(* IEC 61131-3 sources: repolevel_ST_code_completion/extract_code/重型运输系统/modbus/FUN, 16 files *)

(* ---- DataReverse_cmdReverse.st ---- *)
FUNCTION cmdReverse : TargetDirect
VAR_INPUT
	input		:TargetDirect;
END_VAR

IF input = TargetDirect.extend THEN
	cmdReverse := TargetDirect.retract;
END_IF
IF input = TargetDirect.retract THEN
	cmdReverse := TargetDirect.extend;
END_IF

(* ---- percentCalc.st ---- *)
FUNCTION percentCalc : REAL
VAR_INPUT
	level		:INT;	//1->地轨	2->天轨
	idx			:INT;	//挡板索引编号
END_VAR
VAR
	c			:REAL;
	p			:REAL;
END_VAR

//伸出百分比计算
CASE level OF
	1:
		IF gDev.grd[idx].sensor.position < 3 THEN
			RETURN;
		END_IF
		c := gDev.grd[idx].sensor.position - gDev.grd[idx].sensor.retractVal;
		p := gDev.grd[idx].sensor.extendVal - gDev.grd[idx].sensor.retractVal;
		percentCalc := c * 100 / p;
	2:
		IF gDev.sky[idx].sensor.position < 3 THEN
			RETURN;
		END_IF
		c := gDev.sky[idx].sensor.position - gDev.sky[idx].sensor.retractVal;
		p := gDev.sky[idx].sensor.extendVal - gDev.sky[idx].sensor.retractVal;
		percentCalc := c * 100 / p;
END_CASE

(* ---- setButtonByDirect.st ---- *)
FUNCTION setButtonByDirect : BOOL
VAR_INPUT
	level		:INT;	//1->地轨	2->天轨
	idx			:INT;	//挡板索引编号
	direct		:TargetDirect;
END_VAR
VAR
END_VAR
//	本函数用于根据输入参数 操作UI界面的按钮变量
CASE level OF
	1:
		IF idx = 0 OR idx > 10 THEN		//参数校验
			RETURN;
		END_IF
		CASE direct OF
			TargetDirect.extend:
				gUI.grd[idx].btnStop := FALSE;
				gUI.grd[idx].btnExtend := TRUE;
				gUI.grd[idx].btnRetract := FALSE;
			TargetDirect.retract:
				gUI.grd[idx].btnStop := FALSE;
				gUI.grd[idx].btnExtend := FALSE;
				gUI.grd[idx].btnRetract := TRUE;
			TargetDirect.stop:
				gUI.grd[idx].btnStop := FALSE;
				gUI.grd[idx].btnExtend := FALSE;
				gUI.grd[idx].btnRetract := FALSE;
		END_CASE
	2:
		IF idx > 10 THEN		//参数校验
			RETURN;
		END_IF
		CASE direct OF
			TargetDirect.extend:
				gUI.sky[idx].btnStop := FALSE;
				gUI.sky[idx].btnExtend := TRUE;
				gUI.sky[idx].btnRetract := FALSE;
			TargetDirect.retract:
				gUI.sky[idx].btnStop := FALSE;
				gUI.sky[idx].btnExtend := FALSE;
				gUI.sky[idx].btnRetract := TRUE;
			TargetDirect.stop:
				gUI.sky[idx].btnStop := FALSE;
				gUI.sky[idx].btnExtend := FALSE;
				gUI.sky[idx].btnRetract := FALSE;
		END_CASE

END_CASE;

(* ---- updateDevStatus.st ---- *)
FUNCTION updateDevStatus : DevStatus
VAR_INPUT
	level		:INT;		//1->地轨	2->天轨
	idx			:INT;		//挡板索引编号
	errorVal	:REAL;		//误差范围
END_VAR
VAR
	extendVal	:REAL;		//伸出值
	retractVal	:REAL;		//缩回到位值
	nowVal		:REAL;		//当前值
	stat		:DevStatus;	//设备状态
END_VAR

(* 本函数用于根据设备的标定伸出/缩回值以及当前位置
** 判断该缸体是否处于伸出/缩回到位状态，如果到位更新参数
*)

stat := DevStatus.unknown;	//初始化状态量
CASE level OF
	1:
		extendVal := gDev.grd[idx].sensor.extendVal;
		retractVal := gDev.grd[idx].sensor.retractVal;
		nowVal := gDev.grd[idx].sensor.position;
		stat := gDev.grd[idx].state;
	2:
		extendVal := gDev.sky[idx].sensor.extendVal;
		retractVal := gDev.sky[idx].sensor.retractVal;
		nowVal := gDev.sky[idx].sensor.position;
		stat := gDev.sky[idx].state;
END_CASE

IF nowVal > 1 THEN
	IF nowVal < retractVal + errorVal THEN
		stat := DevStatus.retracted;
	ELSIF nowVal > extendVal - errorVal THEN
		stat := DevStatus.extended;
	ELSE
		IF stat <> DevStatus.runing THEN
			stat := DevStatus.error;
		END_IF
	END_IF
ELSE
	stat := DevStatus.unknown;
END_IF

CASE level OF
	1:
		gDev.grd[idx].state := stat;
	2:
		gDev.sky[idx].state := stat;
END_CASE

updateDevStatus := stat;

(* ---- CommandExecutor.st ---- *)
FUNCTION_BLOCK CommandExecutor
VAR_INPUT
	level		:INT;			//1->地轨	2->天轨
	idx			:INT;			//挡板索引编号
	percent		:REAL;			//比例阀百分比 传入-100~+100
END_VAR
VAR_OUTPUT
END_VAR
VAR
END_VAR

IF percent > 0 THEN
	CASE level OF
		1:
			gController.grd[idx].extendPercent := REAL_TO_WORD(percent * 65535 / 100);
			gController.grd[idx].retractPercent := 0;
		2:
			gController.sky[idx].extendPercent := REAL_TO_WORD(percent * 65535 / 100);
			gController.sky[idx].retractPercent := 0;
	END_CASE
ELSE
	CASE level OF
		1:
			gController.grd[idx].extendPercent := 0;
			gController.grd[idx].retractPercent := REAL_TO_WORD(ABS(percent) * 65535 / 100);
		2:
			gController.sky[idx].extendPercent := 0;
			gController.sky[idx].retractPercent := REAL_TO_WORD(ABS(percent) * 65535 / 100);
	END_CASE
END_IF

(* ---- CommandExecutor0.st ---- *)
FUNCTION_BLOCK CommandExecutor0
VAR_INPUT
	level		:INT;			//1->地轨	2->天轨
	idx			:INT;			//挡板索引编号
	direct		:TargetDirect;	//方向
	percent		:REAL;			//比例阀百分比 传入0-100
END_VAR
VAR_OUTPUT
END_VAR
VAR
END_VAR

CASE direct OF
	TargetDirect.extend:
		CASE level OF
			1:
				gController.grd[idx].extendPercent := REAL_TO_WORD(percent * 65535 / 100);
				gController.grd[idx].retractPercent := 0;
			2:
				gController.sky[idx].extendPercent := REAL_TO_WORD(percent * 65535 / 100);
				gController.sky[idx].retractPercent := 0;
		END_CASE
	TargetDirect.retract:
		CASE level OF
			1:
				gController.grd[idx].extendPercent := 0;
				gController.grd[idx].retractPercent := REAL_TO_WORD(percent * 65535 / 100);
			2:
				gController.sky[idx].extendPercent := 0;
				gController.sky[idx].retractPercent := REAL_TO_WORD(percent * 65535 / 100);
		END_CASE
	TargetDirect.stop:
		CASE level OF
			1:
				gController.grd[idx].extendPercent := 0;
				gController.grd[idx].retractPercent := 0;
			2:
				gController.sky[idx].extendPercent := 0;
				gController.sky[idx].retractPercent := 0;
		END_CASE

	ELSE
		CASE level OF
			1:
				gController.grd[idx].extendPercent := 0;
				gController.grd[idx].retractPercent := 0;
			2:
				gController.sky[idx].extendPercent := 0;
				gController.sky[idx].retractPercent := 0;
		END_CASE

END_CASE

(* ---- DataReverse.st ---- *)
FUNCTION_BLOCK DataReverse
VAR_INPUT
END_VAR
VAR_OUTPUT
END_VAR
VAR
END_VAR

(* ---- fileSave.st ---- *)
FUNCTION_BLOCK fileSave
VAR_INPUT
	filePath 	:STRING;
	intervalt	:INT;
END_VAR
VAR
	lineCount	: INT;
	fileHandle  : DWORD;
	fileName	: STRING;
END_VAR
VAR_OUTPUT
END_VAR

(* ---- fileSave_close.st ---- *)
FUNCTION_BLOCK fileSave
VAR_INPUT
	filePath 	:STRING;
	intervalt	:INT;
END_VAR
VAR
	lineCount	: INT;
	fileHandle  : DWORD;
	fileName	: STRING;
END_VAR
VAR_OUTPUT
END_VAR

IF fileHandle <> 0 THEN
	SysFileClose(hFile := fileHandle);
	fileHandle := 0;
END_IF

(* ---- fileSave_createDir.st ---- *)
FUNCTION_BLOCK fileSave
VAR_INPUT
	filePath 	:STRING;
	devName		: STRING ;
	intervalt	:INT;
END_VAR
VAR
	lineCount	: INT;
	fileHandle  : DWORD;
	fileName	: STRING;
	filePath1	:STRING;
END_VAR
VAR_OUTPUT
END_VAR

filePath1 := FilePath;
filePath1 := concat(filePath1,'/');
filePath1 := concat(filePath1,devName);
SysDirCreate2(filePath1, TRUE);

(* ---- fileSave_new.st ---- *)
FUNCTION_BLOCK fileSave
VAR_INPUT
	filePath 	:STRING;
	intervalt	:INT;
	devName		: STRING ;
END_VAR
VAR
	lineCount	: INT;
	fileHandle  : DWORD;
	fileName	: STRING;
	fileHandle0 : DWORD;
	datetime	: DATE_AND_TIME;
	UdIntms 	: UDINT;
	UdMsOffset  : UDINT;
	DTimer_Str  : STRING;
	uiYear 		: UINT;
    uiMonth 	: UINT;
    uiDay 		: UINT;
    uiHour 		: UINT;
    uiMinute 	: UINT;
    uiSecond 	: UINT;
	uiMsSecond	: UINT;

	S_Time64		:  SysTime64;
	STT			:  CurTimeEx;
	S_Time			:  SystemTimeDate;
	Time_Str		:  STRING;
	F_err		: DWORD;
	F_HANDL		: DWORD;
END_VAR
VAR_OUTPUT
END_VAR

	STT(SystemTime:= S_Time64, TimeDate:= S_Time);
	Time_Str :='';
	Time_Str := concat(Time_Str,UINT_TO_STRING(S_Time.Year));
	Time_Str := concat(Time_Str,'-');
	Time_Str := concat(Time_Str,UINT_TO_STRING(S_Time.Month));
	Time_Str := concat(Time_Str,'-');
	Time_Str := concat(Time_Str,UINT_TO_STRING(S_Time.Day));
	Time_Str := concat(Time_Str,'_');
	Time_Str := concat(Time_Str,UINT_TO_STRING(S_Time.Hour));
	Time_Str := concat(Time_Str,'-');
	Time_Str := concat(Time_Str,UINT_TO_STRING(S_Time.Minute));
	Time_Str := concat(Time_Str,'-');
	Time_Str := concat(Time_Str,UINT_TO_STRING(S_Time.Second));
	Time_Str := concat(Time_Str,'_');
	Time_Str := concat(Time_Str,UINT_TO_STRING(S_Time.Milliseconds));

	fileName := FilePath;
	fileName := concat(fileName,'/');
	fileName := concat(fileName,devName);

	fileName := concat(fileName,'/');
	fileName := concat(fileName,devName);
	fileName := concat(fileName,'-');
	fileName := concat(fileName,Time_Str);
    fileName := concat(fileName,'.txt');

	fileHandle := SysFileOpen(szFile:= fileName, am:=ACCESS_MODE.AM_WRITE, pResult:= ADR(F_err));
	lineCount := -1;
	//fileHandle := SysFileOpen(szFile:= fileName, am:=ACCESS_MODE.AM_APPEND, pResult:= ADR(F_err));

(* ---- fileSave_write.st ---- *)
FUNCTION_BLOCK fileSave
VAR_INPUT
	filePath 	:STRING;
	intervalt	:INT;
	positionInt 	:INT;
	speedInt 		:INT;
	stateInt		:INT;
END_VAR
VAR
	lineCount	: INT;
	fileHandle  : DWORD;
	fileName	: STRING;
	data		: STRING;
	F_err		: DWORD;
	tempInt		: INT;
END_VAR
VAR_OUTPUT
END_VAR

IF fileHandle <> 0 THEN
	lineCount := lineCount + 1;
	tempInt	:= lineCount * intervalt;
	data := INT_TO_STRING(lineCount);
	data := concat(data,'$T$T');
	data := concat(data, INT_TO_STRING(tempInt));
	IF tempInt < 1000 THEN
		data := concat(data,'$T');
	END_IF
	data := concat(data,'$T$T');
	data := concat(data,INT_TO_STRING(positionInt));
	data := concat(data,'$T');
	data := concat(data,INT_TO_STRING(speedInt));
	data := concat(data,'$T');
	data := concat(data,INT_TO_STRING(stateInt));
	data := concat(data,'$R');

	SysFileWrite(hFile:=fileHandle , pbyBuffer:= ADR(data) , ulSize:= DINT_TO_DWORD(SysStrLen(data)) , pResult:= ADR(F_err));		// 写入数据

END_IF

(* ---- mdbsLogicToPhy.st ---- *)
FUNCTION_BLOCK mdbsLogicToPhy	//modbus华中挡板地址编号对应本地索引编号
VAR_INPUT
	section		:INT;	//区域限定 1:skyExt, 2:skyRet, 3:grdExt, 4:grdRet)
	lgcIdx		:INT;	//华中对应的地址	10,14{1..10}  17,20{1..11}
END_VAR
VAR_OUTPUT
	level		:INT;	//1->地轨	2->天轨
	phyIdx		:INT;	//内存物理地址对应数组索引
	direct		:TargetDirect;
END_VAR
VAR
END_VAR

(**
 * 将华中指令解析为要动作挡板的标号
 * (level:1->地轨	2->天轨)(phyIdx:内存物理地址对应数组索引)
 *)
CASE section OF
	1://区域限定1:skyExtend)
		level := 2;
		direct := TargetDirect.extend;
		CASE lgcIdx OF
			1:	phyIdx := 1;		//横1	->	sky1
			2:	phyIdx := 3;		//横2	->	sky3
			3:	phyIdx := 4;		//横3	->	sky4
			4:	phyIdx := 5;		//横4	->	sky5
			5:	phyIdx := 6;		//横5	->	sky6
			6:	phyIdx := 8;		//横6	->	sky8
			7:	phyIdx := 9;		//横7	->	sky9
			8:	phyIdx := 10;		//横8	->	sky10
			9:	phyIdx := 2;		//纵1	->	sky2
			10:	phyIdx := 7;		//纵2	->	sky7
			11:	phyIdx := 0;		//起竖	->	sky0
		END_CASE

	2://区域限定2:skyRetract)
		level := 2;
		direct := TargetDirect.retract;
		CASE lgcIdx OF
			1:	phyIdx := 1;		//横1	->	sky1
			2:	phyIdx := 3;		//横2	->	sky3
			3:	phyIdx := 4;		//横3	->	sky4
			4:	phyIdx := 5;		//横4	->	sky5
			5:	phyIdx := 6;		//横5	->	sky6
			6:	phyIdx := 8;		//横6	->	sky8
			7:	phyIdx := 9;		//横7	->	sky9
			8:	phyIdx := 10;		//横8	->	sky10
			9:	phyIdx := 2;		//纵1	->	sky2
			10:	phyIdx := 7;		//纵2	->	sky7
			11:	phyIdx := 0;		//起竖	->	sky0
		END_CASE

	3://区域限定3:grdExtend)
		level := 1;
		direct := TargetDirect.extend;
		CASE lgcIdx OF
			1:	phyIdx := 1;		//横1	->	grd1
			2:	phyIdx := 3;		//横2	->	grd3
			3:	phyIdx := 4;		//横3	->	grd4
			4:	phyIdx := 5;		//横4	->	grd5
			5:	phyIdx := 6;		//横5	->	grd6
			6:	phyIdx := 8;		//横6	->	grd8
			7:	phyIdx := 9;		//横7	->	grd9
			8:	phyIdx := 10;		//横8	->	grd10
			9:	phyIdx := 2;		//纵1	->	grd2
			10:	phyIdx := 7;		//纵2	->	grd7
		END_CASE
	4://区域限定4:grdRetract)
		level := 1;
		direct := TargetDirect.retract;
		CASE lgcIdx OF
			1:	phyIdx := 1;
			2:	phyIdx := 3;
			3:	phyIdx := 4;
			4:	phyIdx := 5;
			5:	phyIdx := 6;
			6:	phyIdx := 8;
			7:	phyIdx := 9;
			8:	phyIdx := 10;
			9:	phyIdx := 2;
			10:	phyIdx := 7;
		END_CASE
END_CASE

(* ---- mdbsNumToIdx.st ---- *)
FUNCTION_BLOCK mdbsNumToIdx
VAR_INPUT
	devNo		:WORD;
END_VAR
VAR_OUTPUT
	level		:INT;
	idx			:INT;
END_VAR
VAR

END_VAR

IF devNo > 40000 THEN
	CASE devNo OF
		//地轨
		41010:	level := 1;	idx := 1;
		41020:	level := 1;	idx := 3;
		41030:	level := 1;	idx := 4;
		41040:	level := 1;	idx := 5;
		41050:	level := 1;	idx := 6;
		41060:	level := 1;	idx := 8;
		41070:	level := 1;	idx := 9;
		41080:	level := 1;	idx := 10;
		42010:	level := 1;	idx := 2;
		42020:	level := 1;	idx := 7;

		51010:	level := 2;	idx := 1;
		51020:	level := 2;	idx := 3;
		51030:	level := 2;	idx := 4;
		51040:	level := 2;	idx := 5;
		51050:	level := 2;	idx := 6;
		51060:	level := 2;	idx := 8;
		51070:	level := 2;	idx := 9;
		51080:	level := 2;	idx := 10;
		52010:	level := 2;	idx := 2;
		52020:	level := 2;	idx := 7;
		53000:	level := 2;	idx := 0;
		53010:	level := 2;	idx := 0;
	END_CASE
END_IF

(* ---- mdbsPhyToLogic.st ---- *)
FUNCTION_BLOCK mdbsPhyToLogic	//modbus本地索引对应回传华中的状态地址
VAR_INPUT
	section		:INT;	//区域限定(1:grdExt, 2:grdRet, 3:skyExt, 4:skyRet)
	phyIdx		:INT;	//内存物理地址对应数组索引
END_VAR
VAR_OUTPUT
	lgcIdx		:INT;	//华中对应的地址	127 175 223 271...
END_VAR
VAR
END_VAR

(**
 * 输入挡板标号，返回华中需要的寄存器地址号
 *)
CASE section OF
	1://区域限定(1:groundExtend)
		CASE phyIdx OF
			1:	lgcIdx := 223;		//grd1e	->	横1	223
			2:	lgcIdx := 231;		//grd2e	->	纵1	231
			3:	lgcIdx := 224;		//grd3e	->	横2	224
			4:	lgcIdx := 225;		//grd4e	->	横3	225
			5:	lgcIdx := 226;		//grd5e	->	横4	226
			6:	lgcIdx := 227;		//grd6e	->	横5	227
			7:	lgcIdx := 232;		//grd7e	->	纵2	232
			8:	lgcIdx := 228;		//grd8e	->	横6	228
			9:	lgcIdx := 229;		//grd9e	->	横7	229
			10:	lgcIdx := 230;		//grd10e->	横8	230
		END_CASE
	2://区域限定(2:groundRetract)
		CASE phyIdx OF
			1:	lgcIdx := 271;		//grd1r	->	横1
			2:	lgcIdx := 279;		//grd2r	->	纵1
			3:	lgcIdx := 272;		//grd3r	->	横2
			4:	lgcIdx := 273;		//grd4r	->	横3
			5:	lgcIdx := 274;		//grd5r	->	横4
			6:	lgcIdx := 275;		//grd6r	->	横5
			7:	lgcIdx := 280;		//grd7r	->	纵2
			8:	lgcIdx := 276;		//grd8r	->	横6
			9:	lgcIdx := 277;		//grd9r	->	横7
			10:	lgcIdx := 278;		//grd10r->	横8
		END_CASE
	3://区域限定(3:skyExtend)
		CASE phyIdx OF
			0:	lgcIdx := 137;		//sky0e	->	起竖
			1:	lgcIdx := 127;		//sky1e	->	横1
			2:	lgcIdx := 135;		//sky2e	->	纵1
			3:	lgcIdx := 128;		//sky3e	->	横2
			4:	lgcIdx := 129;		//sky4e	->	横3
			5:	lgcIdx := 130;		//sky5e	->	横4
			6:	lgcIdx := 131;		//sky6e	->	横5
			7:	lgcIdx := 136;		//sky7e	->	纵2
			8:	lgcIdx := 132;		//sky8e	->	横6
			9:	lgcIdx := 133;		//sky9e	->	横7
			10:	lgcIdx := 134;		//sky10e->	横8
		END_CASE

	4://区域限定(4:skyRetract)
		CASE phyIdx OF
			0:	lgcIdx := 185;		//sky0r	->	起竖
			1:	lgcIdx := 175;		//sky1r	->	横1
			2:	lgcIdx := 183;		//sky2r	->	纵1
			3:	lgcIdx := 176;		//sky3r	->	横2
			4:	lgcIdx := 177;		//sky4r	->	横3
			5:	lgcIdx := 178;		//sky5r	->	横4
			6:	lgcIdx := 179;		//sky6r	->	横5
			7:	lgcIdx := 184;		//sky7r	->	纵2
			8:	lgcIdx := 180;		//sky8r	->	横6
			9:	lgcIdx := 181;		//sky9r	->	横7
			10:	lgcIdx := 182;		//sky10r->	横8
		END_CASE
END_CASE

(* ---- tcpUpload_send.st ---- *)
FUNCTION_BLOCK tcpUpload
VAR_INPUT
	InetAddress		:STRING;
	port			:UINT;
	dataLength		:__XINT;
	sendBuf 		:ARRAY[1..1024]OF BYTE;
END_VAR
VAR_OUTPUT
END_VAR
VAR
	tcpConnector	:TCP.Connector;
	tcpStream		:TCP.Stream;
	pointerStream	:POINTER TO TCP.Stream;
	sizeData		:__XINT;

	tcpState		:UINT:=0;
	tcpCount		:UINT:=0;

	netState		:INT;
END_VAR

tcpCount := tcpCount + 1;
CASE tcpState OF

	0:			//connet server
		tcpConnector.Connect(sIPAddress:= InetAddress,uiPort:= port,pStream => pointerStream);
		IF pointerStream<>0 THEN
			tcpState :=1;
		ELSE
			tcpState :=2;
		END_IF

	1:
		netState := pointerStream^.Send(ADR(sendBuf),dataLength,diSent=>sizeData);
		IF netState <> 0 THEN
			tcpState := 2;
		END_IF

	2:		 	//断开连接
	    tcpConnector.Disconnect();
		tcpState := 0;

END_CASE
